(* This function blocks tests the TEST_FINISHED_NAMED function by creating various tests
   and finishing them in steps *)
FUNCTION_BLOCK FB_TestFinishedNamed EXTENDS TcUnit.FB_TestSuite
VAR
END_VAR

END_FUNCTION_BLOCK

(* stored: Version 1.1.0.1
   POU FB_TestFinishedNamed: Id {845f956b-5469-4f4a-9b3a-de8d813ba965}, SpecialFunc None *)
